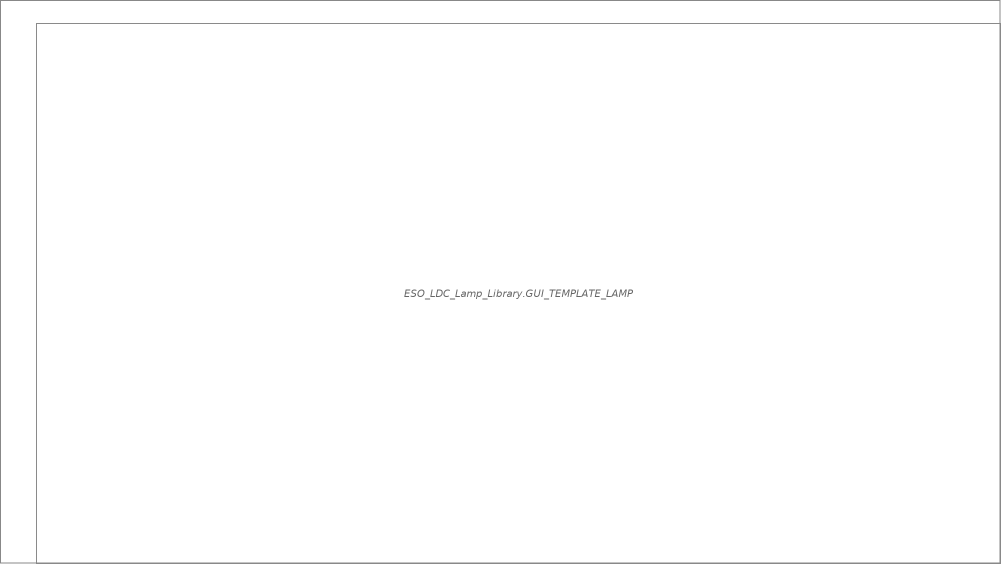
VISUALIZATION lamp1  // 1001x564
    Frame (36,23 965x541)
        shows ESO_LDC_Lamp_Library.GUI_TEMPLATE_LAMP(m_Instance := MAIN.Lamp1)
END_VISUALIZATION

(* stored: Version 1.1.0.1, ProductVersion 3.1.4024.3
   Visu lamp1: Id {1109258a-7deb-4272-bfdf-2cabffbe4465} *)
